FUNCTION_BLOCK RaConnector IMPLEMENTS IService
VAR_INPUT
END_VAR
VAR_OUTPUT
END_VAR
VAR CONSTANT
	TIMEOUT: TIME := T#10S;
END_VAR
VAR
	m_ptrGvlInterface: POINTER TO GvlInterfaceBase;
	m_ptrProcessManager: POINTER TO ProcessManager;
	m_ptrStateTracker: POINTER TO StateTracker;
	m_ptrErrorMgr: POINTER TO ErrorManager;
	
	m_cannotRecover: BOOL;
	m_recoveryRequester: STRING;

	m_recoveryState: ERecoveryState;
	m_conditionToRecover: IExpression;
	m_tonStrategyReceivedTimeout: TON;
	
	m_params : ParameterSet;
	m_alarmId: UINT := 0;
	
	// a store of BoolExpressions that can be assigned at runtime	
	m_boolExpressions: ARRAY [ResiConst.ARR_MIN..ResiConst.COMPENSATIONS_ARR_MAX] OF BoolExpression(0, EBoolOperation.none, 0);
END_VAR

// Specifies that the CPA cannot provide a viable Recovery Strategy.
PROPERTY CannotRecover : BOOL
GET
CannotRecover := m_cannotRecover;
END_GET
END_PROPERTY

METHOD CyclicRaCommunication : BOOL
VAR
	i: UINT;	
	m_ptrCompensation: POINTER TO SCompensation;
	m_ptrRuntimeCond: POINTER TO SRuntimeCondition;
	m_recoveryRes: EOperationResult;
	
	m_count: UINT;
	m_vars: STRING;
	
	m_tmpExpr: IExpression;
	m_valExpr: IValExp;
END_VAR
// OBSERVATION
THIS^.m_ptrGvlInterface^.Out_PtrProcessState := THIS^.m_ptrStateTracker^.PtrProcessState;

// COMPENSATION
m_ptrCompensation := THIS^.m_ptrGvlInterface^.In_PtrCompensations;

FOR i := ResiConst.ARR_MIN TO ResiConst.COMPENSATIONS_ARR_MAX DO
	IF m_ptrCompensation^.IsActive THEN
		CONTINUE;
	END_IF
	
	THIS^.m_ptrGvlInterface^.SetCompensationActive(i, 
		THIS^.m_ptrProcessManager^.Compensate(m_ptrCompensation));
	
	m_ptrCompensation := m_ptrCompensation + SIZEOF(SCompensation);
END_FOR

// RECOVERY
CASE m_recoveryState OF
	ERecoveryState.requested:
		m_cannotRecover := FALSE;
		m_tonStrategyReceivedTimeout(IN := FALSE);
		
		IF m_alarmId = 0 THEN
			// if the requested state is a ValueExpression, it's a request for definition
			IF __QUERYINTERFACE(m_conditionToRecover, m_valExpr) THEN
				m_alarmId := ESpecialAlarmIds.definition_request;
			ELSE
				m_alarmId := ESpecialAlarmIds.recovery_request;
			END_IF
			
			m_ptrErrorMgr^.AddMessage(
				i_alarmId := m_alarmId,
				i_active := TRUE,
				i_severity := ESeverity.warning,
				i_instanceName := m_recoveryRequester);
		END_IF

		// finish all running primitives safely before recovery
		IF m_ptrProcessManager^.FinishPrimitives(i_abortRecoveries := FALSE) THEN
			THIS^.m_ptrGvlInterface^.Out_RecoveryRequestedState := m_conditionToRecover.ToString();
			m_recoveryState := ERecoveryState.awaiting;
			m_alarmId := 0;
		END_IF
		
	ERecoveryState.awaiting:
		m_tonStrategyReceivedTimeout(IN := TRUE, PT := TIMEOUT);
		IF m_tonStrategyReceivedTimeout.Q THEN
			m_recoveryState := ERecoveryState.failed; 
		ELSIF THIS^.m_ptrGvlInterface^.In_RecoveryAvailable THEN
			m_recoveryState := ERecoveryState.running;
		END_IF
		
	// the state is only "failed" if the CPA cannot deliver any viable strategy
	ERecoveryState.failed:
		m_cannotRecover := TRUE;
		m_recoveryState := ERecoveryState.none;
		THIS^.m_ptrGvlInterface^.Out_RecoveryRequestedState := '';
		
	ERecoveryState.running:
		m_recoveryRes := THIS^.m_ptrProcessManager^.ExecuteRecovery(i_strategy := THIS^.m_ptrGvlInterface^.In_Recovery);
		
		// if unsuccessful, the respective primitive has already requested a new recovery
		IF m_recoveryRes = EOperationResult.success THEN
			m_recoveryState := ERecoveryState.completed;
		END_IF
		
	ERecoveryState.completed:
		m_cannotRecover := FALSE;
		m_recoveryState := ERecoveryState.none;
		m_ptrGvlInterface^.ResetRecovery();
END_CASE

// EDITABLE CONDITIONS
m_ptrRuntimeCond := THIS^.m_ptrGvlInterface^.In_PtrRuntimeConditions;
FOR i := ResiConst.ARR_MIN TO ResiConst.COMPENSATIONS_ARR_MAX DO
	IF m_ptrRuntimeCond^.IsActive OR m_ptrRuntimeCond^.PrimitiveId = ESpecialBehaviorIds.empty THEN
		m_ptrRuntimeCond := m_ptrRuntimeCond + SIZEOF(SRuntimeCondition);
		CONTINUE;
	END_IF
	
	m_tmpExpr := GetExpression(m_ptrRuntimeCond^.ExpressionType, m_ptrRuntimeCond^.ExpressionIdx);
	m_ptrProcessManager^.SetPrimitiveCondition(
		m_ptrRuntimeCond^.PrimitiveId, 
		m_ptrRuntimeCond^.IsPre,
		m_tmpExpr);
		
	m_ptrRuntimeCond^.IsActive := TRUE;
	m_ptrRuntimeCond := m_ptrRuntimeCond + SIZEOF(SRuntimeCondition);
END_FOR
END_METHOD

METHOD PRIVATE GetExpression : IExpression
VAR_INPUT
	i_type: EExpressionType;
	i_idx: UINT;
END_VAR
VAR
	m_ptrBoolSpec: POINTER TO SBoolExpressionSpec;
	m_ptrCompExpr: POINTER TO ComparisonExpression;
	m_ptrValExpr: POINTER TO ValueExpression;
END_VAR
CASE i_type OF
	EExpressionType.boolean:
		m_ptrBoolSpec := m_ptrGvlInterface^.In_PtrBoolExprSpecs;
		m_ptrBoolSpec := m_ptrBoolSpec + i_idx * SIZEOF(SBoolExpressionSpec);
		THIS^.m_boolExpressions[i_idx].FB_init(
			FALSE, FALSE,
			i_left := THIS^.GetExpression(m_ptrBoolSpec^.LeftType, m_ptrBoolSpec^.LeftIdx),
			i_sign := m_ptrBoolSpec^.Operator,
			i_right := THIS^.GetExpression(m_ptrBoolSpec^.RightType, m_ptrBoolSpec^.RightIdx));
		GetExpression := THIS^.m_boolExpressions[i_idx];
	
	EExpressionType.comparison:
		m_ptrCompExpr := m_ptrGvlInterface^.In_PtrCompExpressions + i_idx * SIZEOF(ComparisonExpression);
		GetExpression := m_ptrCompExpr^;
	
	EExpressionType.value:
		m_ptrValExpr := m_ptrGvlInterface^.In_PtrValueExpressions + i_idx * SIZEOF(ValueExpression);
		GetExpression := m_ptrValExpr^;
	
	ELSE
		GetExpression := 0;
END_CASE
END_METHOD

METHOD ProvideServices : BOOL
VAR_INPUT
	i_ptrGvlInterface: POINTER TO GvlInterfaceBase;
	i_ptrProcessManager: POINTER TO ProcessManager;
	i_ptrStateTracker: POINTER TO StateTracker;
	i_ptrErrorMgr: POINTER TO ErrorManager;
END_VAR
THIS^.m_ptrGvlInterface := i_ptrGvlInterface;
THIS^.m_ptrProcessManager := i_ptrProcessManager;
THIS^.m_ptrStateTracker := i_ptrStateTracker; 
THIS^.m_ptrErrorMgr := i_ptrErrorMgr;
END_METHOD

PROPERTY RecoveryMode : BOOL
GET
RecoveryMode := m_recoveryState = ERecoveryState.requested
	OR m_recoveryState = ERecoveryState.awaiting
	OR m_recoveryState = ERecoveryState.running
	OR m_recoveryState = ERecoveryState.failed;
END_GET
END_PROPERTY

METHOD RequestRecovery : BOOL
VAR_INPUT
	i_desiredState: IExpression;
	i_senderName: STRING;
END_VAR
// "recursive" recoveries are not supported
IF m_recoveryState <> ERecoveryState.none THEN
	RETURN;
END_IF

m_recoveryState := ERecoveryState.requested;
m_conditionToRecover := i_desiredState;
m_recoveryRequester := i_senderName;
END_METHOD

END_FUNCTION_BLOCK

(* stored: Version 1.1.0.1, ProductVersion 3.1.4024.12
   POU RaConnector: Id {7e7193e1-8358-4bce-ad37-62ecd9b52c8e}, SpecialFunc None
   Property CannotRecover: Id {b5dfec31-9fe6-44ee-9dd9-90068c7c7b60}
   Get Get: Id {ea84626a-02f7-4273-a28f-2c62e7a856c9}
   Method CyclicRaCommunication: Id {044b793f-c721-4bee-826e-85cf5fc55473}
   Method GetExpression: Id {dc273b51-6231-4bac-b35d-98f32c342612}
   Method ProvideServices: Id {0dbc4ec7-0bf8-4a7e-a7b7-98ea2eefb342}
   Property RecoveryMode: Id {eae8ec6d-4a3d-4d3a-a01f-0da6d6f8348c}
   Get Get: Id {2e97f02f-44c5-4182-95c8-1c31aa2fb382}
   Method RequestRecovery: Id {811befea-5cad-42ce-b233-09231cb46c78} *)
